FUNCTION_BLOCK SENSOR_UBI_MQTT_V2
  {SET_ATTRIBUTE(OpcUa, SERVICE)}
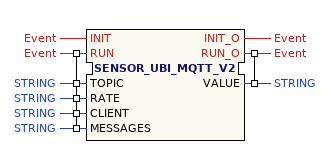
  EVENT_INPUT
    INIT;
    RUN WITH TOPIC, RATE, CLIENT, MESSAGES;
  END_EVENT
  EVENT_OUTPUT
    INIT_O;
    RUN_O WITH VALUE;
  END_EVENT
  VAR_INPUT
    TOPIC : STRING; {SET_ATTRIBUTE(OpcUa, Constant)}
    RATE : STRING; {SET_ATTRIBUTE(OpcUa, Constant)}
    CLIENT : STRING; {SET_ATTRIBUTE(OpcUa, Variable)}
    MESSAGES : STRING; {SET_ATTRIBUTE(OpcUa, Variable)}
  END_VAR
  VAR_OUTPUT
    VALUE : STRING; {SET_ATTRIBUTE(OpcUa, Variable)}
  END_VAR
END_FUNCTION_BLOCK
